{attribute 'pack_mode' := '1'}
TYPE MoveAxisRelative EXTENDS IncomingMessage :
STRUCT
	axisIndex: INT; (* 1 or 2.*)
	distance: LREAL;
	moveTime: TIME;
END_STRUCT
END_TYPE

(* stored: Version 1.1.0.1, ProductVersion 3.1.4022.12
   DUT MoveAxisRelative: Id {ea912ee2-7216-4c72-8b01-91a2f30753f0} *)
